// TIA Portal V18 export
FUNCTION_BLOCK "nokButtonQUE"   // FB10, LAD
{ S7_Optimized_Access := 'TRUE' }
VERSION : 0.1
// stored: AutoNumber true, IsIECCheckEnabled false, IsRetainMemResEnabled false, MemoryReserve 100, SetENOAutomatically false, UDAEnableTagReadback false
   VAR_OUTPUT
      O_nokPart : Bool;
   END_VAR
   VAR_IN_OUT
      buttonQue : Int;
   END_VAR
   VAR
      "step" : Byte;
      TIM_countOn { S7_SetPoint := 'True'} : TON_TIME;
      TIM_countOff { S7_SetPoint := 'True'} : TON_TIME;
      countOn : Bool;
      countOff : Bool;
   END_VAR
BEGIN

REGION Network 1: Jump List
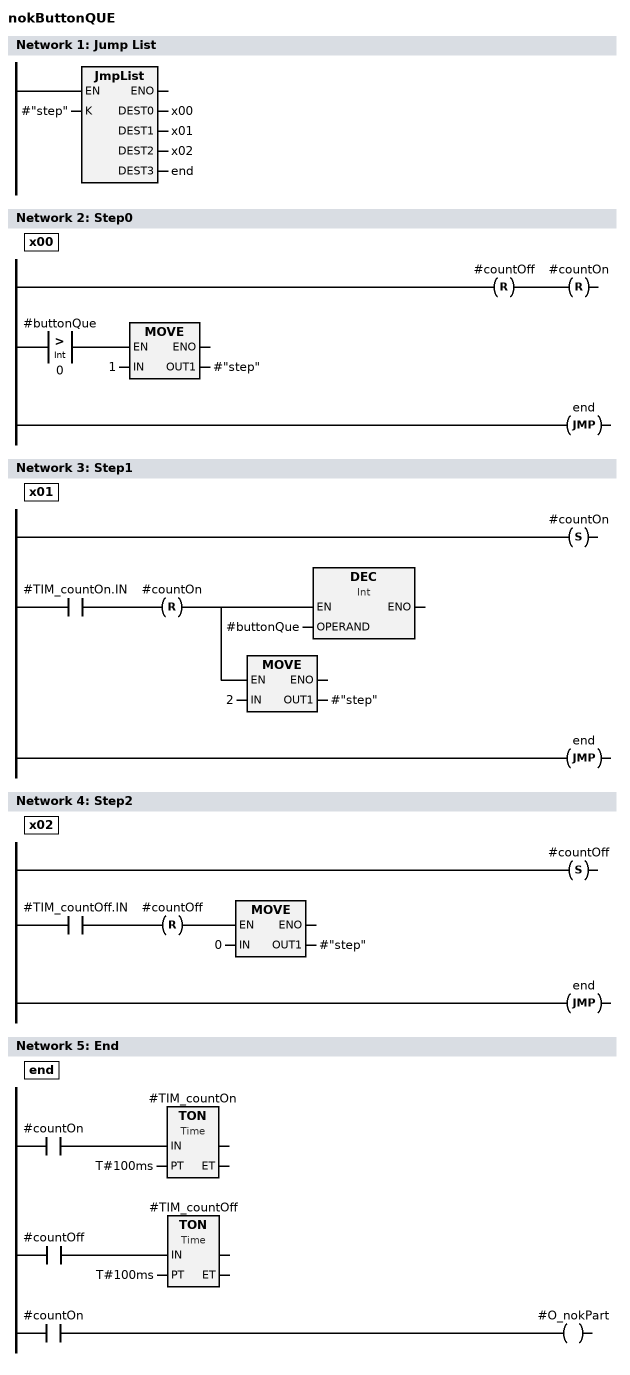
   // no SCL statement known for JmpList: written as a call
   JmpList(k := #"step", dest0 => x00, dest1 => x01, dest2 => x02, dest3 => end);
END_REGION

REGION Network 2: Step0
   Label( x00 )
   RUNG wire#powerrail
      R_Coil( #countOff )
      R_Coil( #countOn )
   END_RUNG
   RUNG wire#powerrail
      { S7_Templates := "SrcType := Int" } GT_Contact(in1 := #buttonQue, in2 := 0)
      Move(in := 1, out1 => #"step")
   END_RUNG
   RUNG wire#powerrail
      JumpCoil( end )
   END_RUNG
   // the same network as SCL:
   x00:
   #countOff := FALSE;
   #countOn := FALSE;
   IF #buttonQue > 0 THEN #"step" := 1; END_IF;
   GOTO end;
END_REGION

REGION Network 3: Step1
   Label( x01 )
   RUNG wire#powerrail
      S_Coil( #countOn )
   END_RUNG
   RUNG wire#powerrail
      Contact( #TIM_countOn.IN )
      R_Coil( #countOn )
      wire#w1
      { S7_Templates := "DestType := Int" } Dec( #buttonQue )
   END_RUNG
   RUNG wire#w1
      Move(in := 2, out1 => #"step")
   END_RUNG
   RUNG wire#powerrail
      JumpCoil( end )
   END_RUNG
   // the same network as SCL:
   x01:
   #countOn := TRUE;
   IF #TIM_countOn.IN THEN
       #countOn := FALSE;
       #buttonQue := #buttonQue - 1;
       #"step" := 2;
   END_IF;
   GOTO end;
END_REGION

REGION Network 4: Step2
   Label( x02 )
   RUNG wire#powerrail
      S_Coil( #countOff )
   END_RUNG
   RUNG wire#powerrail
      Contact( #TIM_countOff.IN )
      R_Coil( #countOff )
      Move(in := 0, out1 => #"step")
   END_RUNG
   RUNG wire#powerrail
      JumpCoil( end )
   END_RUNG
   // the same network as SCL:
   x02:
   #countOff := TRUE;
   IF #TIM_countOff.IN THEN
       #countOff := FALSE;
       #"step" := 0;
   END_IF;
   GOTO end;
END_REGION

REGION Network 5: End
   Label( end )
   RUNG wire#powerrail
      Contact( #countOn )
      { S7_Templates := "time_type := Time" } #TIM_countOn.TON(pt := T#100ms, et =>)
   END_RUNG
   RUNG wire#powerrail
      Contact( #countOff )
      { S7_Templates := "time_type := Time" } #TIM_countOff.TON(pt := T#100ms, et =>)
   END_RUNG
   RUNG wire#powerrail
      Contact( #countOn )
      Coil( #O_nokPart )
   END_RUNG
   // the same network as SCL:
   end:
   #TIM_countOn(IN := #countOn, PT := T#100ms);   // TON
   #TIM_countOff(IN := #countOff, PT := T#100ms);   // TON
   #O_nokPart := #countOn;
END_REGION
END_FUNCTION_BLOCK
